Universal Robots PolyScope program: edges_dev.urp

Program edges_dev (installation=cube_dev1 directory=/programs/cube createdIn=5.11.5.1010327 lastSavedIn=5.11.5.1010327 robotSerialNumber=20215500677)
Calibrated DH parameters: a=[0.000204, -0.239222, -0.391845, -0.000001, 0.000022, 0]; d=[0.162722, -355.808559, 353.37206, 2.570385, 0.099741, 0.099629]; alpha=[1.571124, 0.000988, 0.008295, 1.568963, -1.570303, 0]; deltaTheta=[0, -0.973091, 7.204745, 0.05153, 0, 0]
Robot Program (runOnlyOnce=true)
  MoveJ speed 60 deg/s, acceleration 80 deg/s^2 (useActiveTCP=false) tcp=SandTCP; feature=Base
    Waypoint Waypoint (Variable): variable(featureName=edges_origin)
  MoveJ speed 60 deg/s, acceleration 80 deg/s^2 (useActiveTCP=true) feature=Base
    Waypoint Waypoint_1 (Relative): relativeFromPosition TCP in base x=499.982 y=-100.008 z=100.019 mm, rx=1.2085 ry=1.2095 rz=1.2086 rad; joints [131.502, -68.712, 131.039, -6.124, 58.056, -38.248] deg; TCP offset x=1.003 y=125.541 z=104.154 mm, rx=-0.7854 ry=0 rz=0 rad; TCP in base x=499.978 y=-100.016 z=99.984 mm, rx=1.4817 ry=0.6145 rz=0.6132 rad; joints [167.832, -65.327, 122.332, -6.929, 112.593, 24.835] deg
  MoveL speed 100 mm/s, acceleration 1200 mm/s^2 (useActiveTCP=false) tcp=SprayTCP; feature=Base
    MoveDirectionNode (selectedDirection=ZPlus)
      Until DISTANCE (allowActions=false deceleration=3 distanceNodeType=BLEND) Distance=0.365; motionParameters(blendRadius=0.025)
    MoveDirectionNode (selectedDirection=ZMinus) feature=Joint_6_name
      Until DISTANCE (allowActions=false deceleration=3 distanceNodeType=STOP) Distance=0.1; motionParameters(blendRadius=0)
    MoveJ speed 60 deg/s, acceleration 80 deg/s^2 (useActiveTCP=true) feature=Base
      Waypoint Waypoint_2 (Relative): relativeFromPosition TCP in base x=525.019 y=-200.014 z=565.481 mm, rx=0.6137 ry=1.4822 rz=-0.6139 rad; joints [161.097, -90.845, 79.166, 12.516, 160.933, -89.104] deg; TCP in base x=525.003 y=-200.035 z=565.453 mm, rx=0 ry=2.3562 rz=0 rad; joints [138.093, -75.297, 36.925, 68.976, 100.608, -118.77] deg
    MoveDirectionNode (selectedDirection=YMinus)
      Until DISTANCE (allowActions=false deceleration=3 distanceNodeType=BLEND) Distance=0.365; motionParameters(blendRadius=0.025)
    MoveDirectionNode (selectedDirection=ZMinus)
      Until DISTANCE (allowActions=false deceleration=3 distanceNodeType=BLEND) Distance=0.365; motionParameters(blendRadius=0.025)
    MoveDirectionNode (selectedDirection=YPlus)
      Until DISTANCE (allowActions=false deceleration=3 distanceNodeType=BLEND) Distance=0.365; motionParameters(blendRadius=0.025)
